// TIA Portal project "Handling_and_Signal_Conditioning" (V15.1)

(* hardware
DEVICE "S7-1200 station_1"  S7-1200 Station
   slot 0: "Rack_0"  S7-1200 Rack  Rack  V1.0
   slot 1: "PLC_1"  CPU 1214C DC/DC/DC  6ES7 214-1AG40-0XB0  V4.2
*)

// ===== PLC "PLC_1"  CPU 1214C DC/DC/DC =====

VAR_GLOBAL   // PLC tag table "Default tag table"
   "Start_Switch" AT %M0.0 : Bool;
   "Prox_Sensor" AT %M0.1 : Bool;
   "Edge_Mem" AT %M0.2 : Bool;
   "Parts_Count" AT %MW20 : Int;
   "Total_Weight" AT %MD24 : Real;
   "Parts_Real_Temp" AT %MD28 : Real;
END_VAR

ORGANIZATION_BLOCK "Main"   // OB1, LAD, ProgramCycle
TITLE = "Main Program Sweep (Cycle)"
{ S7_Optimized_Access := 'TRUE' }
VERSION : 0.1
   VAR_INPUT
      Initial_Call : Bool;   // Initial call of this OB
      Remanence : Bool;   // =True, if remanent data are available
   END_VAR
   VAR_TEMP   // added for the SCL form of the ladder/FBD networks
      _w1 : Bool;
      _w2 : Bool;
   END_VAR
BEGIN

REGION Network 1
   // Production Counter Logic: Increments the total parts count (%MW20) by 1 using a rising edge pulse (P_TRIG) from the proximity sensor (%M0.1) only when the system start switch (%M0.0) is active. This prevents double-counting if a part stalls in front of the sensor
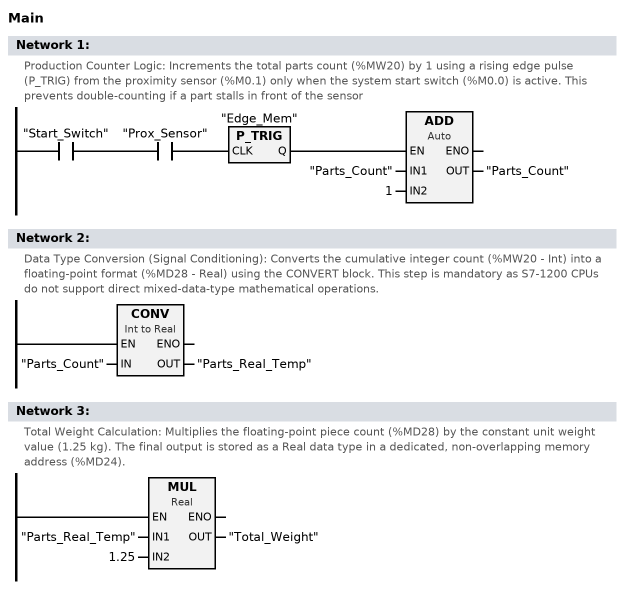
   RUNG wire#powerrail
      Contact( "Start_Switch" )
      Contact( "Prox_Sensor" )
      P_Trig( "Edge_Mem" )
      Add(in1 := "Parts_Count", in2 := 1, out => "Parts_Count")
   END_RUNG
   // the same network as SCL:
   #_w1 := "Start_Switch" AND "Prox_Sensor";
   #_w2 := #_w1 AND NOT "Edge_Mem";   // rising edge
   "Edge_Mem" := #_w1;
   IF #_w2 THEN "Parts_Count" := "Parts_Count" + 1; END_IF;
END_REGION

REGION Network 2
   // Data Type Conversion (Signal Conditioning): Converts the cumulative integer count (%MW20 - Int) into a floating-point format (%MD28 - Real) using the CONVERT block. This step is mandatory as S7-1200 CPUs do not support direct mixed-data-type mathematical operations.
   RUNG wire#powerrail
      { S7_Templates := "[SrcType := Int, DestType := Real]" } Convert(in := "Parts_Count", out => "Parts_Real_Temp")
   END_RUNG
   // the same network as SCL:
   "Parts_Real_Temp" := INT_TO_REAL("Parts_Count");
END_REGION

REGION Network 3
   // Total Weight Calculation: Multiplies the floating-point piece count (%MD28) by the constant unit weight value (1.25 kg). The final output is stored as a Real data type in a dedicated, non-overlapping memory address (%MD24).
   RUNG wire#powerrail
      { S7_Templates := "SrcType := Real" } Mul(in1 := "Parts_Real_Temp", in2 := 1.25, out => "Total_Weight")
   END_RUNG
   // the same network as SCL:
   "Total_Weight" := "Parts_Real_Temp" * 1.25;
END_REGION
END_ORGANIZATION_BLOCK